FUNCTION_BLOCK FB_Elevator_SFC EXTENDS FB_Object_Template_SFC
VAR_INPUT

//Señales de accion
	Up:BOOL;
	Down:BOOL;
	Step:BOOL;
	
//Finales de carrera
	END_Up:BOOL;
	END_Down:BOOL;
	END_Step:BOOL;

END_VAR
VAR_OUTPUT
	
//Acciones
	MOV_Up:BOOL;
	MOV_Down:BOOL;
	MOV_Step:BOOL;

END_VAR
VAR
	
	T :TIME := T#0.5S;

END_VAR

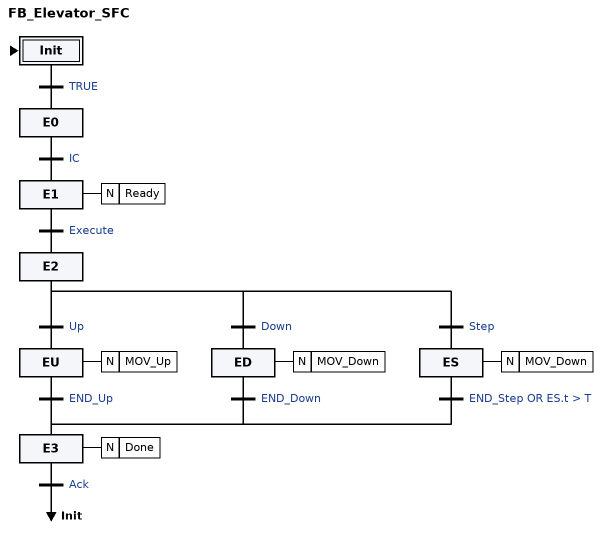
INITIAL_STEP Init:
END_STEP
TRANSITION FROM Init TO E0
    := TRUE;
END_TRANSITION
STEP E0:
END_STEP
TRANSITION FROM E0 TO E1
    := IC;
END_TRANSITION
STEP E1:
    Ready(N);
END_STEP
TRANSITION FROM E1 TO E2
    := Execute;
END_TRANSITION
STEP E2:
END_STEP
TRANSITION FROM E2 TO EU
    := Up;
END_TRANSITION
STEP EU:
    MOV_Up(N);
END_STEP
TRANSITION FROM EU TO E3
    := END_Up;
END_TRANSITION
TRANSITION FROM E2 TO ED
    := Down;
END_TRANSITION
STEP ED:
    MOV_Down(N);
END_STEP
TRANSITION FROM ED TO E3
    := END_Down;
END_TRANSITION
TRANSITION FROM E2 TO ES
    := Step;
END_TRANSITION
STEP ES:
    MOV_Down(N);
END_STEP
TRANSITION FROM ES TO E3
    := END_Step OR ES.t > T;
END_TRANSITION
STEP E3:
    Done(N);
END_STEP
TRANSITION FROM E3 TO Init
    := Ack;
END_TRANSITION

TRANSITION Execute:
Up OR Down OR Step;
END_TRANSITION

END_FUNCTION_BLOCK

(* stored: Version 1.1.0.1, ProductVersion 3.1.4024.6
   POU FB_Elevator_SFC: Id {d1da8d57-d49f-4b70-b3c5-3cd810f5a6c4}, SpecialFunc None
   Transition Execute: Id {d2a2dd6d-f778-48ef-9083-e2d7915d0a83} *)
